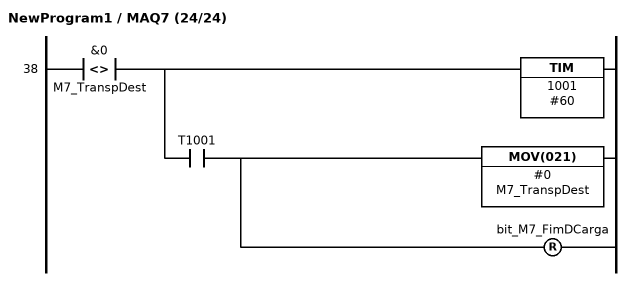
; [picture p24: NewProgram1 / MAQ7, rungs 38-38]
; rung 38
LD<>(305) &0 M7_TranspDest
TIM 1001 #60
AND T1001
MOV(021) #0 M7_TranspDest
RSET bit_M7_FimDCarga

### Section MAQ8

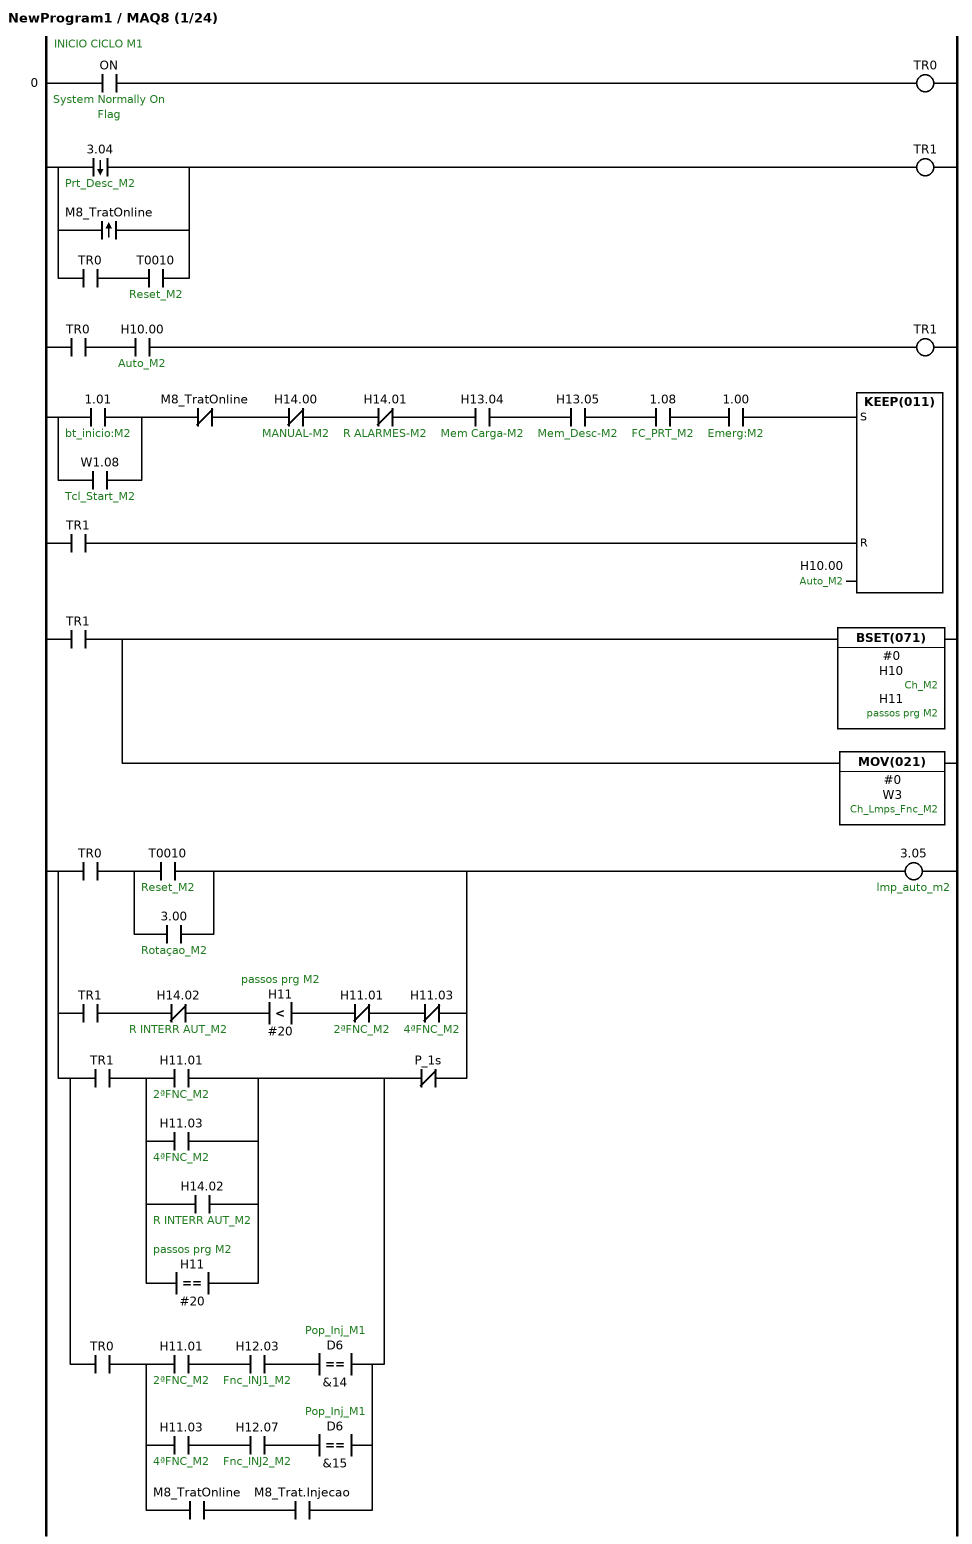
; rung 0: INICIO CICLO M1
LD 1.01  ; bt_inicio:M2
OR W1.08  ; Tcl_Start_M2
ANDNOT M8_TratOnline
ANDNOT H14.00  ; MANUAL-M2
ANDNOT H14.01  ; R ALARMES-M2
AND H13.04  ; Mem Carga-M2
AND H13.05  ; Mem_Desc-M2
AND 1.08  ; FC_PRT_M2
AND 1.00  ; Emerg:M2
%LD 3.04  ; Prt_Desc_M2
@OR M8_TratOnline
LD ON  ; System Normally On Flag
OUT TR0
AND T0010  ; Reset_M2
ORLD
OUT TR1
KEEP(011) H10.00  ; Auto_M2
LD TR1
BSET(071) #0 H10 H11  ; Ch_M2, passos prg M2
MOV(021) #0 W3  ; Ch_Lmps_Fnc_M2
LD TR0
LD T0010  ; Reset_M2
OR 3.00  ; Rotaçao_M2
ANDLD
LD TR0
AND H10.00  ; Auto_M2
OUT TR1
ANDNOT H14.02  ; R INTERR AUT_M2
AND<(310) H11 #20  ; passos prg M2
ANDNOT H11.01  ; 2ªFNC_M2
ANDNOT H11.03  ; 4ªFNC_M2
ORLD
LD TR1
LD H11.01  ; 2ªFNC_M2
OR H11.03  ; 4ªFNC_M2
OR H14.02  ; R INTERR AUT_M2
OR=(300) H11 #20  ; passos prg M2
ANDLD
LD TR0
LD H11.01  ; 2ªFNC_M2
AND H12.03  ; Fnc_INJ1_M2
AND=(300) D6 &14  ; Pop_Inj_M1
LD H11.03  ; 4ªFNC_M2
AND H12.07  ; Fnc_INJ2_M2
AND=(300) D6 &15  ; Pop_Inj_M1
ORLD
LD M8_TratOnline
AND M8_Trat.Injecao
ORLD
ANDLD
ORLD
ANDNOT P_1s
ORLD
OUT 3.05  ; lmp_auto_m2

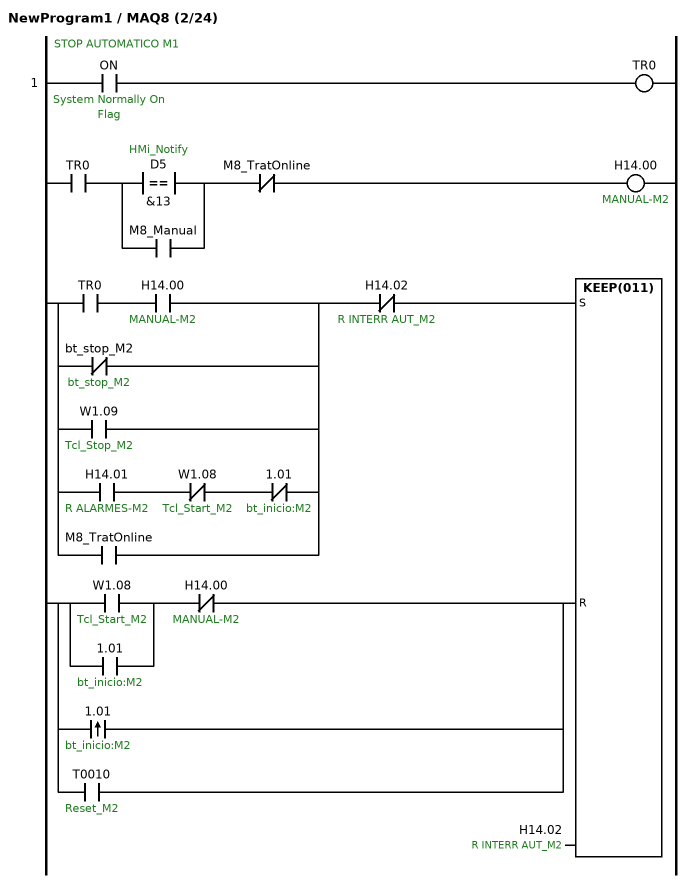
; rung 1: STOP AUTOMATICO M1
LD ON  ; System Normally On Flag
OUT TR0
LD=L(301) D5 &13  ; HMi_Notify
OR M8_Manual
ANDLD
ANDNOT M8_TratOnline
OUT H14.00  ; MANUAL-M2
LD TR0
AND H14.00  ; MANUAL-M2
LDNOT bt_stop_M2  ; bt_stop_M2
OR W1.09  ; Tcl_Stop_M2
LD H14.01  ; R ALARMES-M2
ANDNOT W1.08  ; Tcl_Start_M2
ANDNOT 1.01  ; bt_inicio:M2
ORLD
OR M8_TratOnline
ORLD
ANDNOT H14.02  ; R INTERR AUT_M2
LD W1.08  ; Tcl_Start_M2
OR 1.01  ; bt_inicio:M2
ANDNOT H14.00  ; MANUAL-M2
@OR 1.01  ; bt_inicio:M2
OR T0010  ; Reset_M2
KEEP(011) H14.02  ; R INTERR AUT_M2

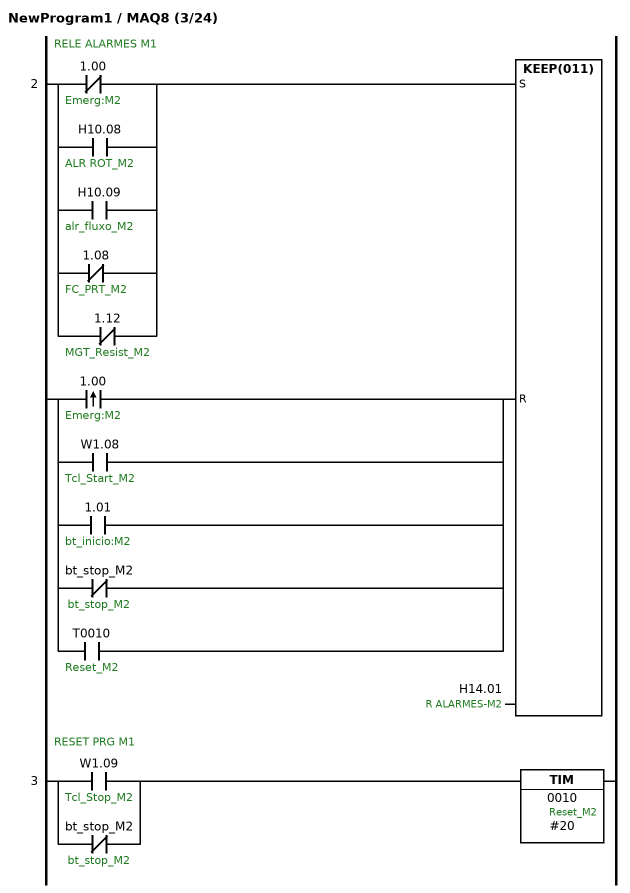
; rung 2: RELE ALARMES M1
LDNOT 1.00  ; Emerg:M2
OR H10.08  ; ALR ROT_M2
OR H10.09  ; alr_fluxo_M2
ORNOT 1.08  ; FC_PRT_M2
ORNOT 1.12  ; MGT_Resist_M2
@LD 1.00  ; Emerg:M2
OR W1.08  ; Tcl_Start_M2
OR 1.01  ; bt_inicio:M2
ORNOT bt_stop_M2  ; bt_stop_M2
OR T0010  ; Reset_M2
KEEP(011) H14.01  ; R ALARMES-M2
; rung 3: RESET PRG M1
LD W1.09  ; Tcl_Stop_M2
ORNOT bt_stop_M2  ; bt_stop_M2
TIM 0010 #20  ; Reset_M2

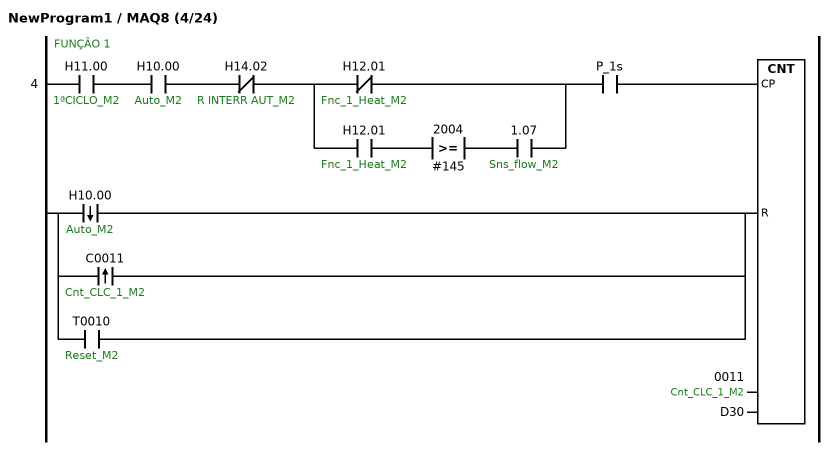
; rung 4: FUNÇÂO 1
LD H11.00  ; 1ªCICLO_M2
AND H10.00  ; Auto_M2
ANDNOT H14.02  ; R INTERR AUT_M2
LDNOT H12.01  ; Fnc_1_Heat_M2
LD H12.01  ; Fnc_1_Heat_M2
AND>=(325) 2004 #145
AND 1.07  ; Sns_flow_M2
ORLD
ANDLD
AND P_1s
%LD H10.00  ; Auto_M2
@OR C0011  ; Cnt_CLC_1_M2
OR T0010  ; Reset_M2
CNT 0011 D30  ; Cnt_CLC_1_M2

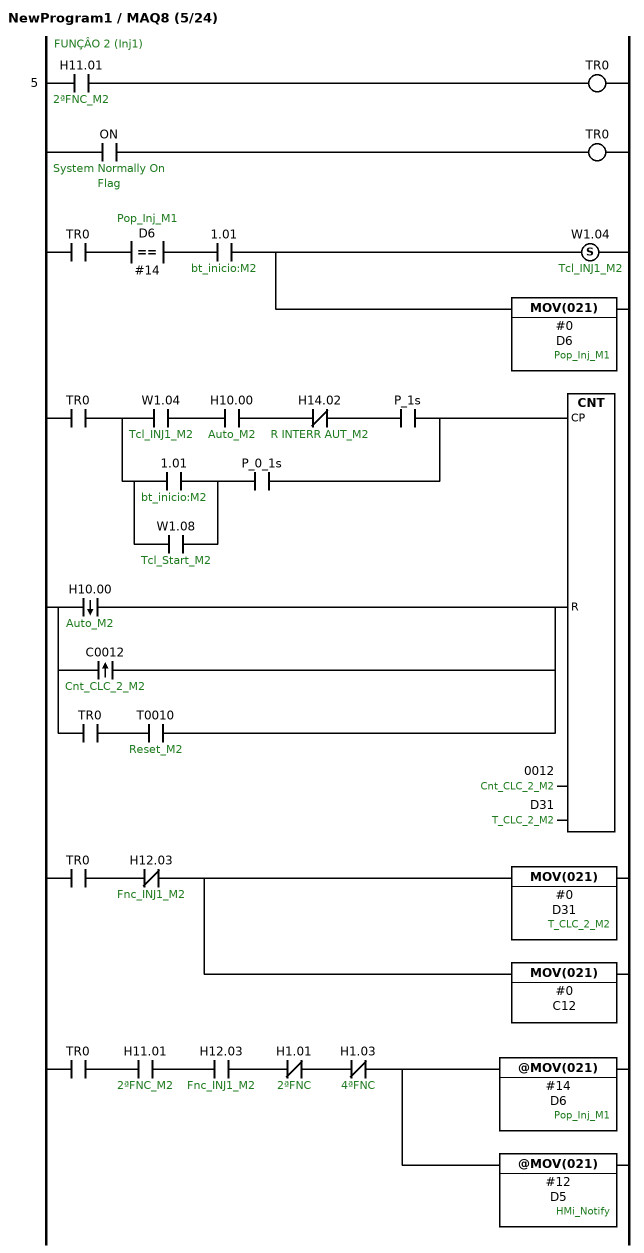
; rung 5: FUNÇÂO 2 (Inj1)
LD H11.01  ; 2ªFNC_M2
OUT TR0
AND=(300) D6 #14  ; Pop_Inj_M1
AND 1.01  ; bt_inicio:M2
SET W1.04  ; Tcl_INJ1_M2
MOV(021) #0 D6  ; Pop_Inj_M1
LD TR0
LD W1.04  ; Tcl_INJ1_M2
AND H10.00  ; Auto_M2
ANDNOT H14.02  ; R INTERR AUT_M2
AND P_1s
LD 1.01  ; bt_inicio:M2
OR W1.08  ; Tcl_Start_M2
AND P_0_1s
ORLD
ANDLD
%LD H10.00  ; Auto_M2
@OR C0012  ; Cnt_CLC_2_M2
LD ON  ; System Normally On Flag
OUT TR0
AND T0010  ; Reset_M2
ORLD
CNT 0012 D31  ; T_CLC_2_M2, Cnt_CLC_2_M2
LD TR0
ANDNOT H12.03  ; Fnc_INJ1_M2
MOV(021) #0 D31  ; T_CLC_2_M2
MOV(021) #0 C12
LD TR0
AND H11.01  ; 2ªFNC_M2
AND H12.03  ; Fnc_INJ1_M2
ANDNOT H1.01  ; 2ªFNC
ANDNOT H1.03  ; 4ªFNC
@MOV(021) #14 D6  ; Pop_Inj_M1
@MOV(021) #12 D5  ; HMi_Notify

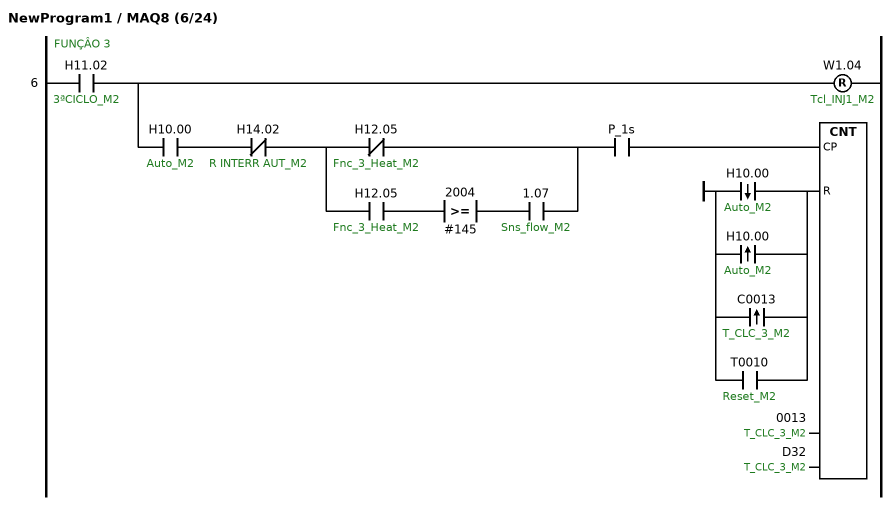
; rung 6: FUNÇÂO 3
LD H11.02  ; 3ªCICLO_M2
RSET W1.04  ; Tcl_INJ1_M2
AND H10.00  ; Auto_M2
ANDNOT H14.02  ; R INTERR AUT_M2
LDNOT H12.05  ; Fnc_3_Heat_M2
LD H12.05  ; Fnc_3_Heat_M2
AND>=(325) 2004 #145
AND 1.07  ; Sns_flow_M2
ORLD
ANDLD
AND P_1s
%LD H10.00  ; Auto_M2
@OR H10.00  ; Auto_M2
@OR C0013  ; T_CLC_3_M2
OR T0010  ; Reset_M2
CNT 0013 D32  ; T_CLC_3_M2

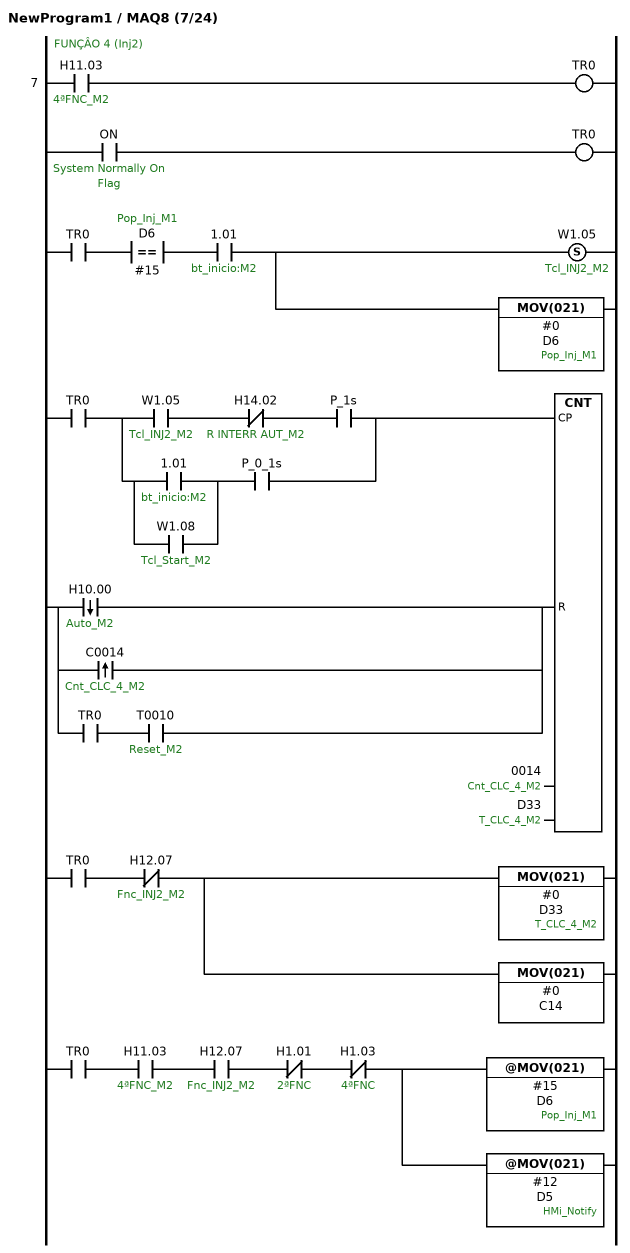
; rung 7: FUNÇÂO 4 (Inj2)
LD H11.03  ; 4ªFNC_M2
OUT TR0
AND=(300) D6 #15  ; Pop_Inj_M1
AND 1.01  ; bt_inicio:M2
SET W1.05  ; Tcl_INJ2_M2
MOV(021) #0 D6  ; Pop_Inj_M1
LD TR0
LD W1.05  ; Tcl_INJ2_M2
ANDNOT H14.02  ; R INTERR AUT_M2
AND P_1s
LD 1.01  ; bt_inicio:M2
OR W1.08  ; Tcl_Start_M2
AND P_0_1s
ORLD
ANDLD
%LD H10.00  ; Auto_M2
@OR C0014  ; Cnt_CLC_4_M2
LD ON  ; System Normally On Flag
OUT TR0
AND T0010  ; Reset_M2
ORLD
CNT 0014 D33  ; T_CLC_4_M2, Cnt_CLC_4_M2
LD TR0
ANDNOT H12.07  ; Fnc_INJ2_M2
MOV(021) #0 D33  ; T_CLC_4_M2
MOV(021) #0 C14
LD TR0
AND H11.03  ; 4ªFNC_M2
AND H12.07  ; Fnc_INJ2_M2
ANDNOT H1.01  ; 2ªFNC
ANDNOT H1.03  ; 4ªFNC
@MOV(021) #15 D6  ; Pop_Inj_M1
@MOV(021) #12 D5  ; HMi_Notify

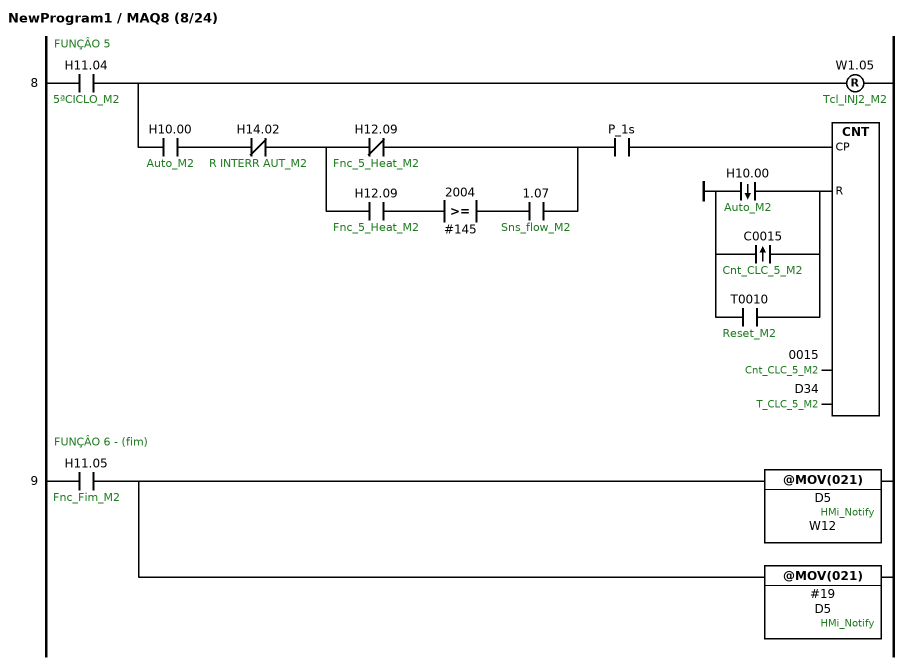
; rung 8: FUNÇÂO 5
LD H11.04  ; 5ªCICLO_M2
RSET W1.05  ; Tcl_INJ2_M2
AND H10.00  ; Auto_M2
ANDNOT H14.02  ; R INTERR AUT_M2
LDNOT H12.09  ; Fnc_5_Heat_M2
LD H12.09  ; Fnc_5_Heat_M2
AND>=(325) 2004 #145
AND 1.07  ; Sns_flow_M2
ORLD
ANDLD
AND P_1s
%LD H10.00  ; Auto_M2
@OR C0015  ; Cnt_CLC_5_M2
OR T0010  ; Reset_M2
CNT 0015 D34  ; T_CLC_5_M2, Cnt_CLC_5_M2
; rung 9: FUNÇÂO 6 - (fim)
LD H11.05  ; Fnc_Fim_M2
@MOV(021) D5 W12  ; HMi_Notify
@MOV(021) #19 D5  ; HMi_Notify

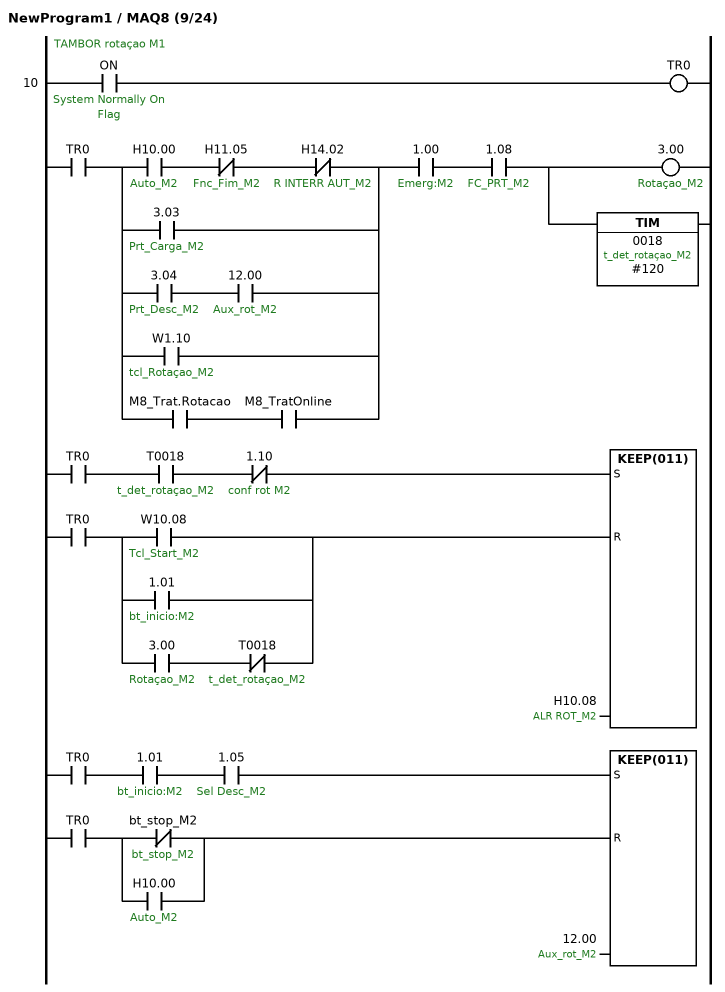
; rung 10: TAMBOR rotaçao M1
LD ON  ; System Normally On Flag
OUT TR0
LD H10.00  ; Auto_M2
ANDNOT H11.05  ; Fnc_Fim_M2
ANDNOT H14.02  ; R INTERR AUT_M2
OR 3.03  ; Prt_Carga_M2
LD 3.04  ; Prt_Desc_M2
AND 12.00  ; Aux_rot_M2
ORLD
OR W1.10  ; tcl_Rotaçao_M2
LD M8_Trat.Rotacao
AND M8_TratOnline
ORLD
ANDLD
AND 1.00  ; Emerg:M2
AND 1.08  ; FC_PRT_M2
OUT 3.00  ; Rotaçao_M2
TIM 0018 #120  ; t_det_rotaçao_M2
LD TR0
AND T0018  ; t_det_rotaçao_M2
ANDNOT 1.10  ; conf rot M2
LD TR0
LD W10.08  ; Tcl_Start_M2
OR 1.01  ; bt_inicio:M2
LD 3.00  ; Rotaçao_M2
ANDNOT T0018  ; t_det_rotaçao_M2
ORLD
ANDLD
KEEP(011) H10.08  ; ALR ROT_M2
LD TR0
AND 1.01  ; bt_inicio:M2
AND 1.05  ; Sel Desc_M2
LD TR0
LDNOT bt_stop_M2  ; bt_stop_M2
OR H10.00  ; Auto_M2
ANDLD
KEEP(011) 12.00  ; Aux_rot_M2

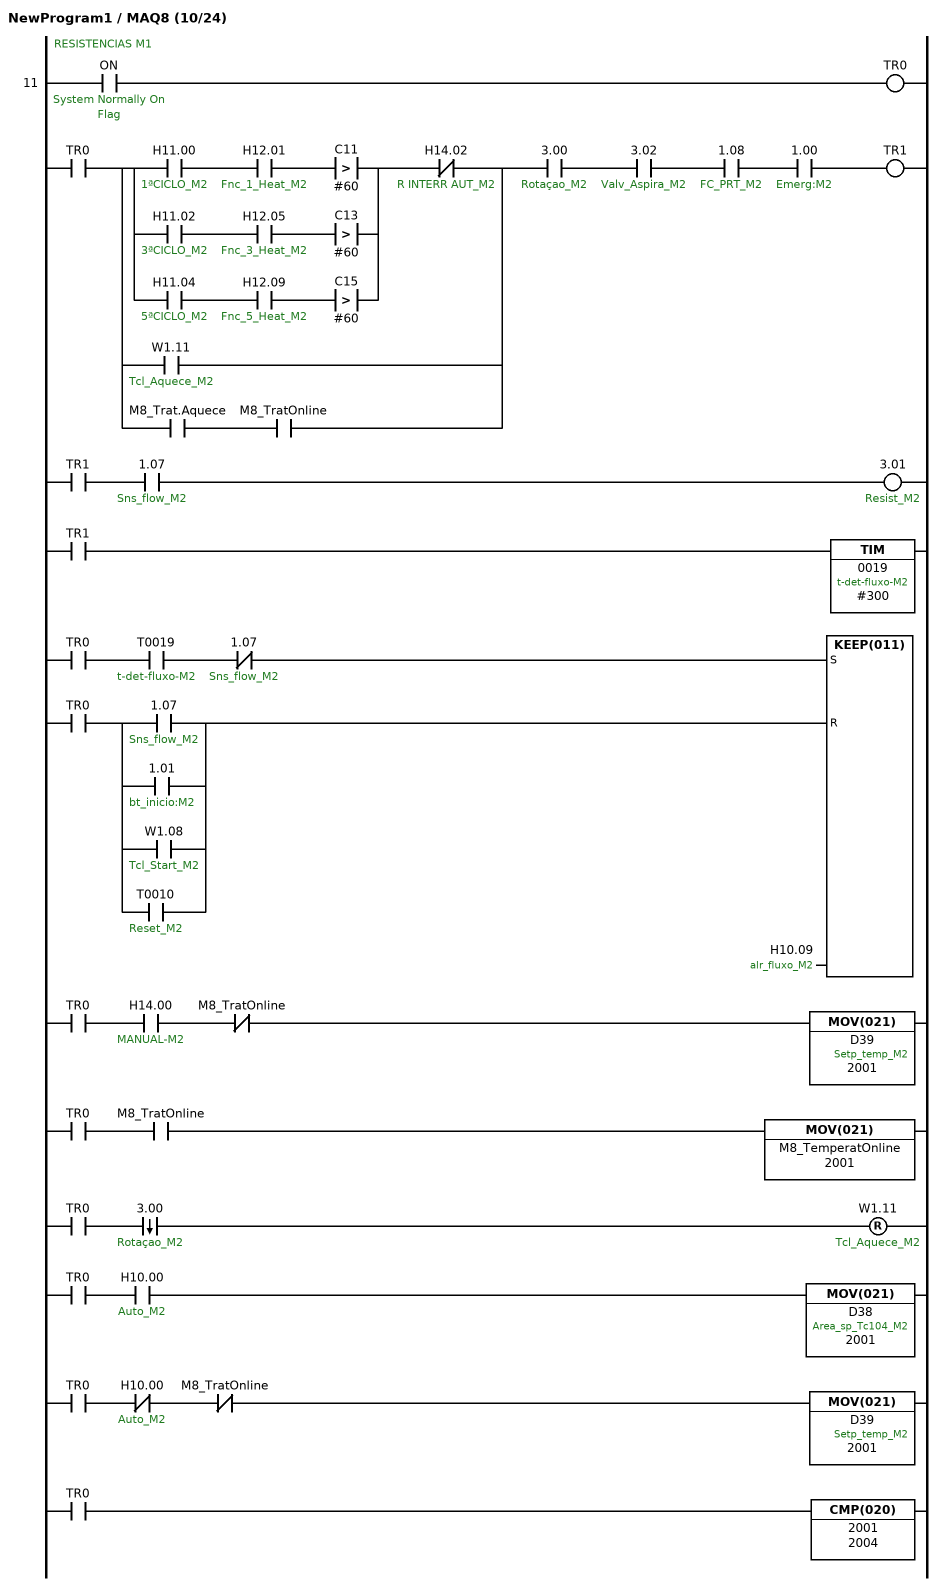
; rung 11: RESISTENCIAS M1
LD ON  ; System Normally On Flag
OUT TR0
LD H11.00  ; 1ªCICLO_M2
AND H12.01  ; Fnc_1_Heat_M2
AND>(320) C11 #60
LD H11.02  ; 3ªCICLO_M2
AND H12.05  ; Fnc_3_Heat_M2
AND>(320) C13 #60
ORLD
LD H11.04  ; 5ªCICLO_M2
AND H12.09  ; Fnc_5_Heat_M2
AND>(320) C15 #60
ORLD
ANDNOT H14.02  ; R INTERR AUT_M2
OR W1.11  ; Tcl_Aquece_M2
LD M8_Trat.Aquece
AND M8_TratOnline
ORLD
ANDLD
AND 3.00  ; Rotaçao_M2
AND 3.02  ; Valv_Aspira_M2
AND 1.08  ; FC_PRT_M2
AND 1.00  ; Emerg:M2
OUT TR1
AND 1.07  ; Sns_flow_M2
OUT 3.01  ; Resist_M2
LD TR1
TIM 0019 #300  ; t-det-fluxo-M2
LD TR0
AND T0019  ; t-det-fluxo-M2
ANDNOT 1.07  ; Sns_flow_M2
LD TR0
LD 1.07  ; Sns_flow_M2
OR 1.01  ; bt_inicio:M2
OR W1.08  ; Tcl_Start_M2
OR T0010  ; Reset_M2
ANDLD
KEEP(011) H10.09  ; alr_fluxo_M2
LD TR0
AND H14.00  ; MANUAL-M2
ANDNOT M8_TratOnline
MOV(021) D39 2001  ; Setp_temp_M2
LD TR0
AND M8_TratOnline
MOV(021) M8_TemperatOnline 2001
LD TR0
%AND 3.00  ; Rotaçao_M2
RSET W1.11  ; Tcl_Aquece_M2
LD TR0
AND H10.00  ; Auto_M2
MOV(021) D38 2001  ; Area_sp_Tc104_M2
LD TR0
ANDNOT H10.00  ; Auto_M2
ANDNOT M8_TratOnline
MOV(021) D39 2001  ; Setp_temp_M2
LD TR0
CMP(020) 2001 2004

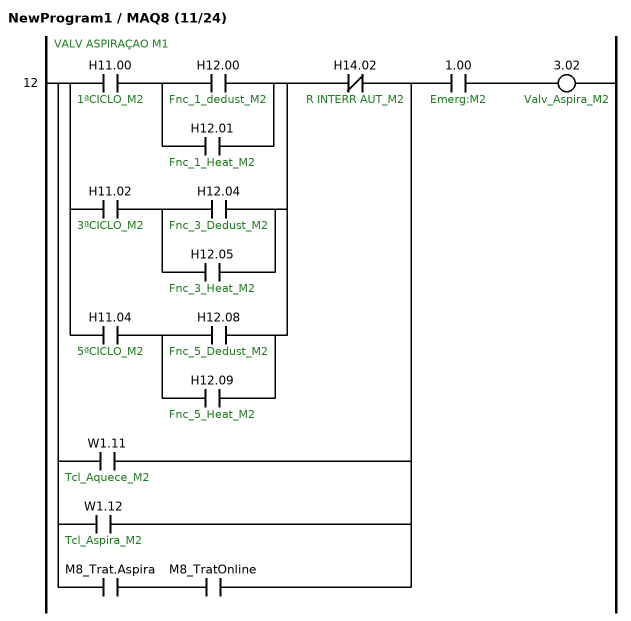
; rung 12: VALV ASPIRAÇAO M1
LD H11.00  ; 1ªCICLO_M2
LD H12.00  ; Fnc_1_dedust_M2
OR H12.01  ; Fnc_1_Heat_M2
ANDLD
LD H11.02  ; 3ªCICLO_M2
LD H12.04  ; Fnc_3_Dedust_M2
OR H12.05  ; Fnc_3_Heat_M2
ANDLD
ORLD
LD H11.04  ; 5ªCICLO_M2
LD H12.08  ; Fnc_5_Dedust_M2
OR H12.09  ; Fnc_5_Heat_M2
ANDLD
ORLD
ANDNOT H14.02  ; R INTERR AUT_M2
OR W1.11  ; Tcl_Aquece_M2
OR W1.12  ; Tcl_Aspira_M2
LD M8_Trat.Aspira
AND M8_TratOnline
ORLD
AND 1.00  ; Emerg:M2
OUT 3.02  ; Valv_Aspira_M2

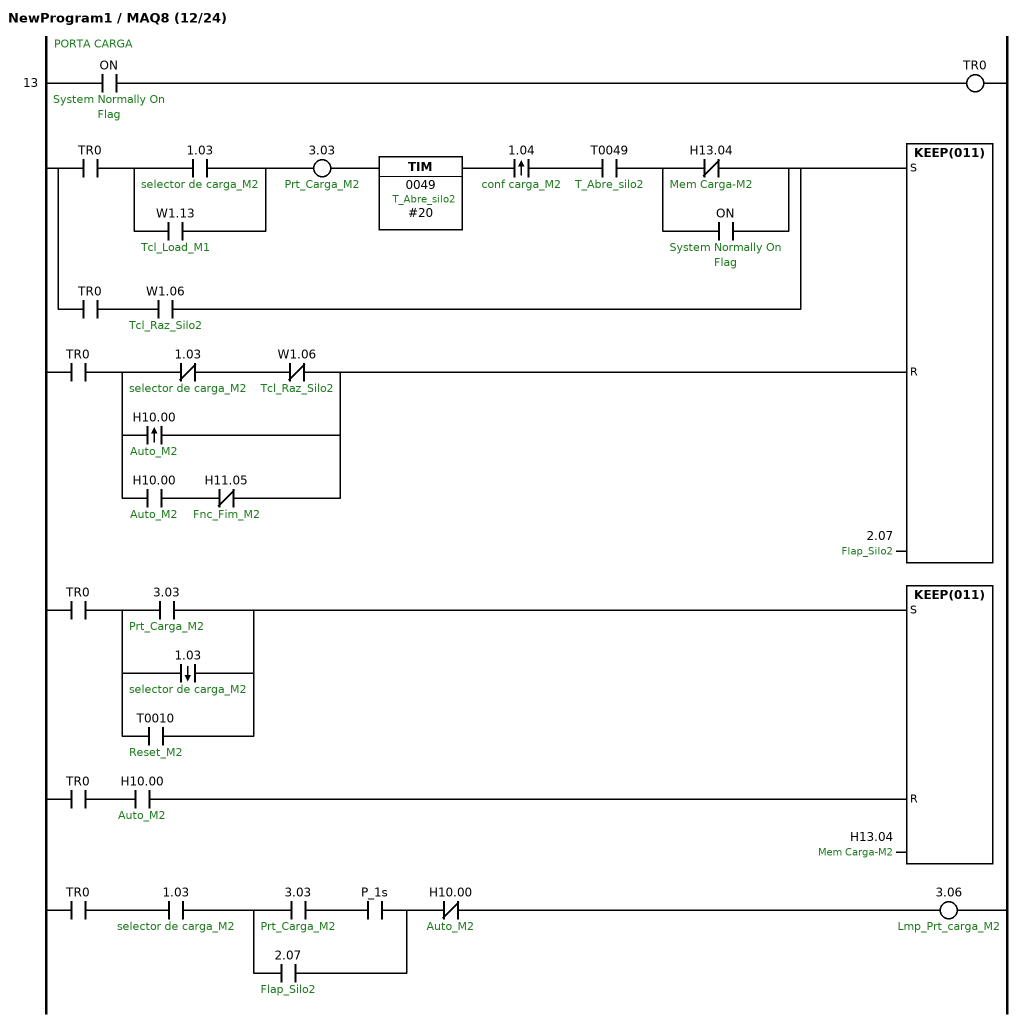
; rung 13: PORTA CARGA
LD ON  ; System Normally On Flag
OUT TR0
LD 1.03  ; selector de carga_M2
OR W1.13  ; Tcl_Load_M1
ANDLD
OUT 3.03  ; Prt_Carga_M2
TIM 0049 #20  ; T_Abre_silo2
@AND 1.04  ; conf carga_M2
AND T0049  ; T_Abre_silo2
LDNOT H13.04  ; Mem Carga-M2
OR ON  ; System Normally On Flag
ANDLD
LD TR0
AND W1.06  ; Tcl_Raz_Silo2
ORLD
LD TR0
LDNOT 1.03  ; selector de carga_M2
ANDNOT W1.06  ; Tcl_Raz_Silo2
@OR H10.00  ; Auto_M2
LD H10.00  ; Auto_M2
ANDNOT H11.05  ; Fnc_Fim_M2
ORLD
ANDLD
KEEP(011) 2.07  ; Flap_Silo2
LD TR0
LD 3.03  ; Prt_Carga_M2
%OR 1.03  ; selector de carga_M2
OR T0010  ; Reset_M2
ANDLD
LD TR0
AND H10.00  ; Auto_M2
KEEP(011) H13.04  ; Mem Carga-M2
LD TR0
AND 1.03  ; selector de carga_M2
LD 3.03  ; Prt_Carga_M2
AND P_1s
OR 2.07  ; Flap_Silo2
ANDLD
ANDNOT H10.00  ; Auto_M2
OUT 3.06  ; Lmp_Prt_carga_M2

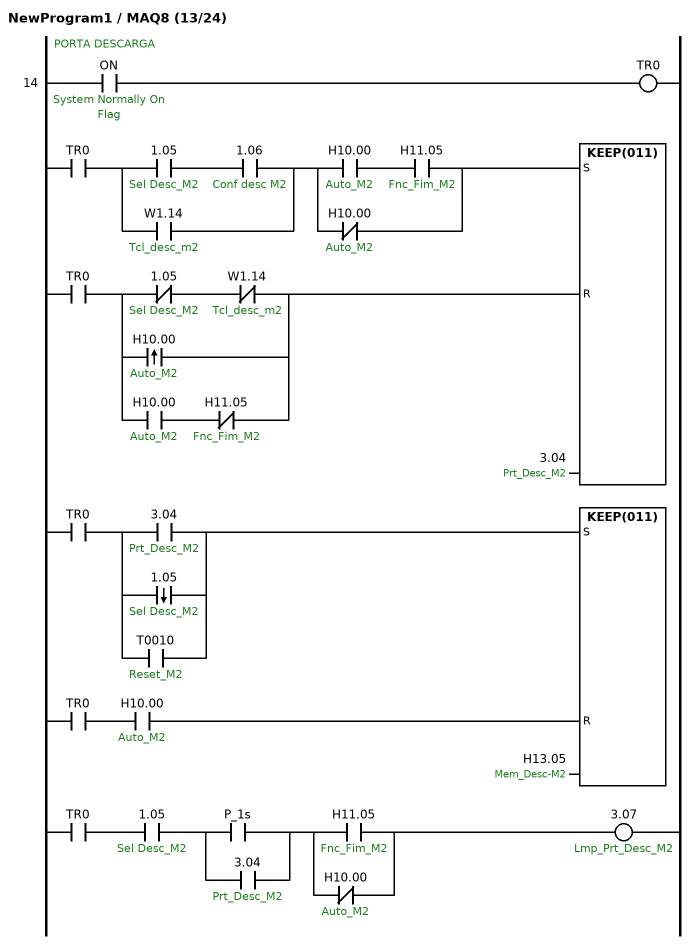
; rung 14: PORTA DESCARGA
LD ON  ; System Normally On Flag
OUT TR0
LD 1.05  ; Sel Desc_M2
AND 1.06  ; Conf desc M2
OR W1.14  ; Tcl_desc_m2
ANDLD
LD H10.00  ; Auto_M2
AND H11.05  ; Fnc_Fim_M2
ORNOT H10.00  ; Auto_M2
ANDLD
LD TR0
LDNOT 1.05  ; Sel Desc_M2
ANDNOT W1.14  ; Tcl_desc_m2
@OR H10.00  ; Auto_M2
LD H10.00  ; Auto_M2
ANDNOT H11.05  ; Fnc_Fim_M2
ORLD
ANDLD
KEEP(011) 3.04  ; Prt_Desc_M2
LD TR0
LD 3.04  ; Prt_Desc_M2
%OR 1.05  ; Sel Desc_M2
OR T0010  ; Reset_M2
ANDLD
LD TR0
AND H10.00  ; Auto_M2
KEEP(011) H13.05  ; Mem_Desc-M2
LD TR0
AND 1.05  ; Sel Desc_M2
LD P_1s
OR 3.04  ; Prt_Desc_M2
ANDLD
LD H11.05  ; Fnc_Fim_M2
ORNOT H10.00  ; Auto_M2
ANDLD
OUT 3.07  ; Lmp_Prt_Desc_M2

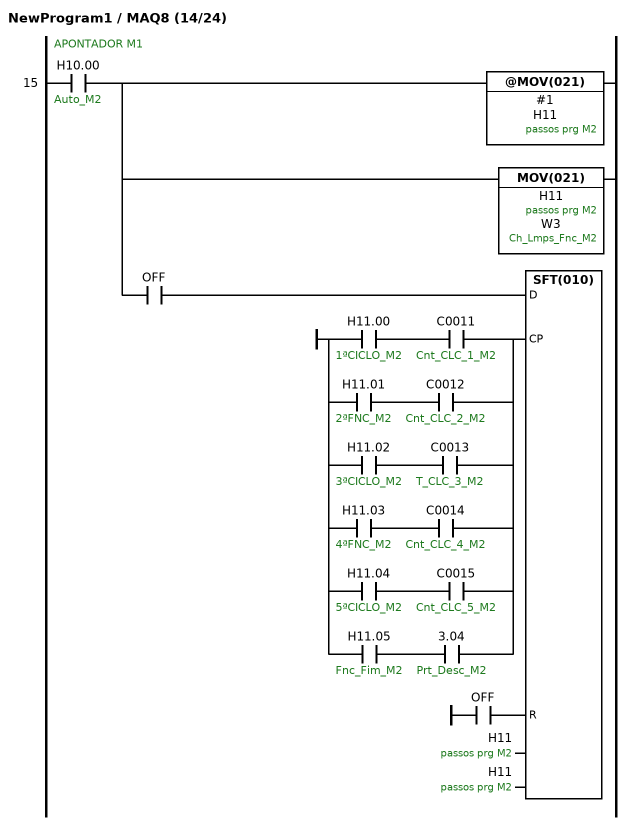
; rung 15: APONTADOR M1
LD H10.00  ; Auto_M2
@MOV(021) #1 H11  ; passos prg M2
MOV(021) H11 W3  ; passos prg M2, Ch_Lmps_Fnc_M2
AND OFF
LD H11.00  ; 1ªCICLO_M2
AND C0011  ; Cnt_CLC_1_M2
LD H11.01  ; 2ªFNC_M2
AND C0012  ; Cnt_CLC_2_M2
ORLD
LD H11.02  ; 3ªCICLO_M2
AND C0013  ; T_CLC_3_M2
ORLD
LD H11.03  ; 4ªFNC_M2
AND C0014  ; Cnt_CLC_4_M2
ORLD
LD H11.04  ; 5ªCICLO_M2
AND C0015  ; Cnt_CLC_5_M2
ORLD
LD H11.05  ; Fnc_Fim_M2
AND 3.04  ; Prt_Desc_M2
ORLD
LD OFF
SFT(010) H11 H11  ; passos prg M2

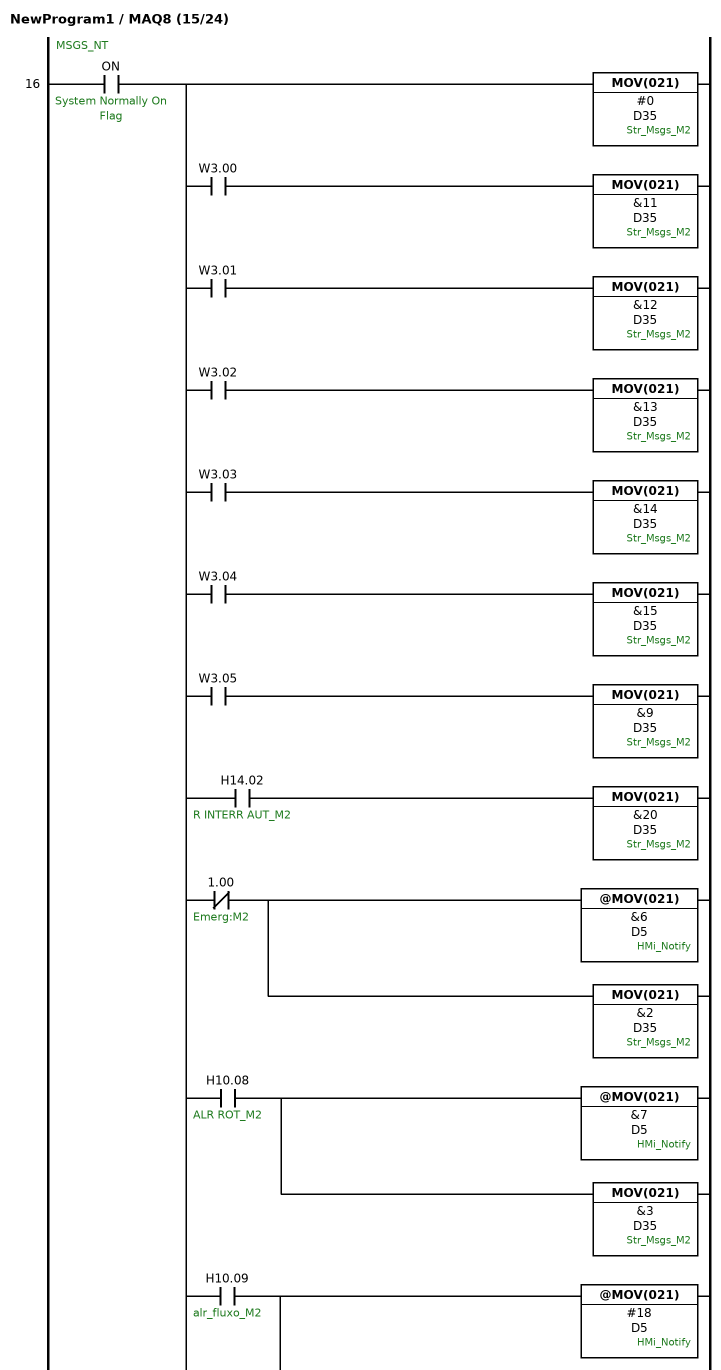

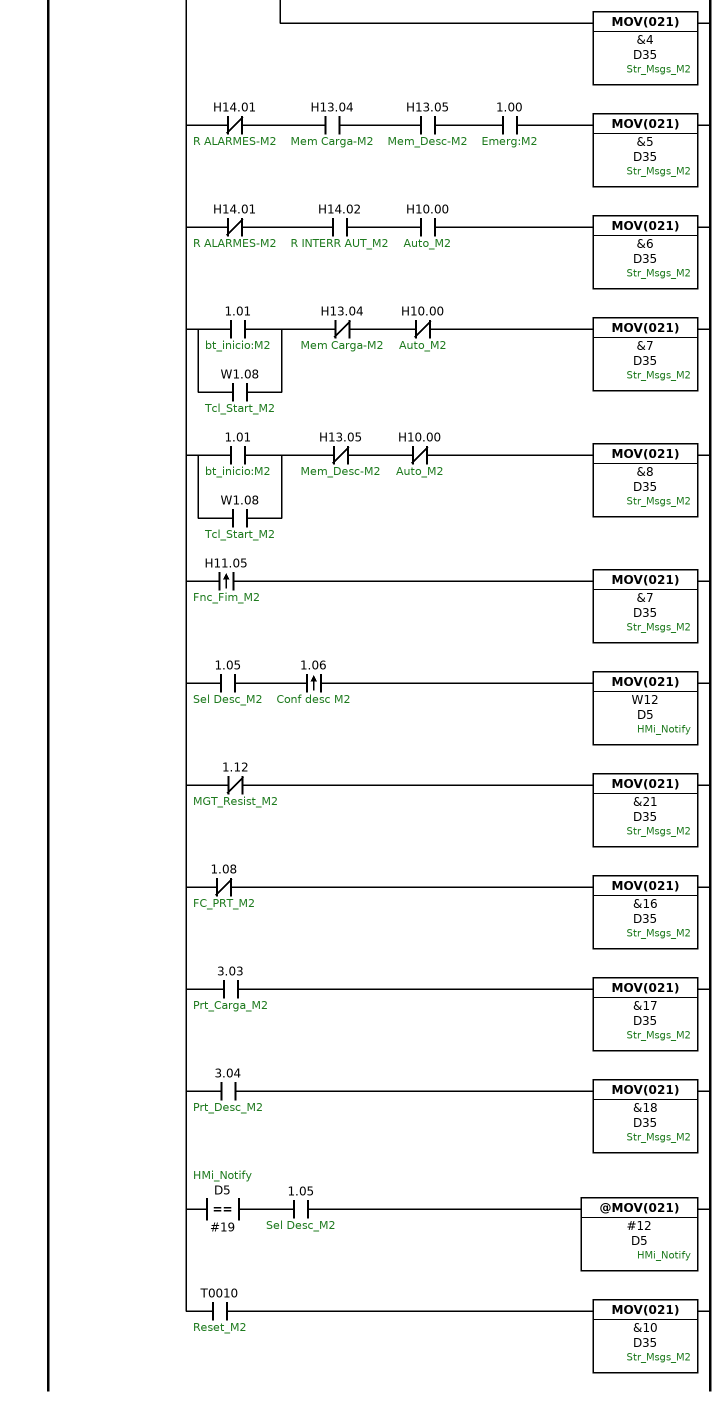
; rung 16: MSGS_NT
LD ON  ; System Normally On Flag
OUT TR0
MOV(021) #0 D35  ; Str_Msgs_M2
AND W3.00
MOV(021) &11 D35  ; Str_Msgs_M2
LD TR0
AND W3.01
MOV(021) &12 D35  ; Str_Msgs_M2
LD TR0
AND W3.02
MOV(021) &13 D35  ; Str_Msgs_M2
LD TR0
AND W3.03
MOV(021) &14 D35  ; Str_Msgs_M2
LD TR0
AND W3.04
MOV(021) &15 D35  ; Str_Msgs_M2
LD TR0
AND W3.05
MOV(021) &9 D35  ; Str_Msgs_M2
LD TR0
AND H14.02  ; R INTERR AUT_M2
MOV(021) &20 D35  ; Str_Msgs_M2
LD TR0
ANDNOT 1.00  ; Emerg:M2
@MOV(021) &6 D5  ; HMi_Notify
MOV(021) &2 D35  ; Str_Msgs_M2
LD TR0
AND H10.08  ; ALR ROT_M2
@MOV(021) &7 D5  ; HMi_Notify
MOV(021) &3 D35  ; Str_Msgs_M2
LD TR0
AND H10.09  ; alr_fluxo_M2
@MOV(021) #18 D5  ; HMi_Notify
MOV(021) &4 D35  ; Str_Msgs_M2
LD TR0
ANDNOT H14.01  ; R ALARMES-M2
AND H13.04  ; Mem Carga-M2
AND H13.05  ; Mem_Desc-M2
AND 1.00  ; Emerg:M2
MOV(021) &5 D35  ; Str_Msgs_M2
LD TR0
ANDNOT H14.01  ; R ALARMES-M2
AND H14.02  ; R INTERR AUT_M2
AND H10.00  ; Auto_M2
MOV(021) &6 D35  ; Str_Msgs_M2
LD TR0
LD 1.01  ; bt_inicio:M2
OR W1.08  ; Tcl_Start_M2
ANDLD
ANDNOT H13.04  ; Mem Carga-M2
ANDNOT H10.00  ; Auto_M2
MOV(021) &7 D35  ; Str_Msgs_M2
LD TR0
LD 1.01  ; bt_inicio:M2
OR W1.08  ; Tcl_Start_M2
ANDLD
ANDNOT H13.05  ; Mem_Desc-M2
ANDNOT H10.00  ; Auto_M2
MOV(021) &8 D35  ; Str_Msgs_M2
LD TR0
@AND H11.05  ; Fnc_Fim_M2
MOV(021) &7 D35  ; Str_Msgs_M2
LD TR0
AND 1.05  ; Sel Desc_M2
@AND 1.06  ; Conf desc M2
MOV(021) W12 D5  ; HMi_Notify
LD TR0
ANDNOT 1.12  ; MGT_Resist_M2
MOV(021) &21 D35  ; Str_Msgs_M2
LD TR0
ANDNOT 1.08  ; FC_PRT_M2
MOV(021) &16 D35  ; Str_Msgs_M2
LD TR0
AND 3.03  ; Prt_Carga_M2
MOV(021) &17 D35  ; Str_Msgs_M2
LD TR0
AND 3.04  ; Prt_Desc_M2
MOV(021) &18 D35  ; Str_Msgs_M2
LD TR0
AND=(300) D5 #19  ; HMi_Notify
AND 1.05  ; Sel Desc_M2
@MOV(021) #12 D5  ; HMi_Notify
LD TR0
AND T0010  ; Reset_M2
MOV(021) &10 D35  ; Str_Msgs_M2

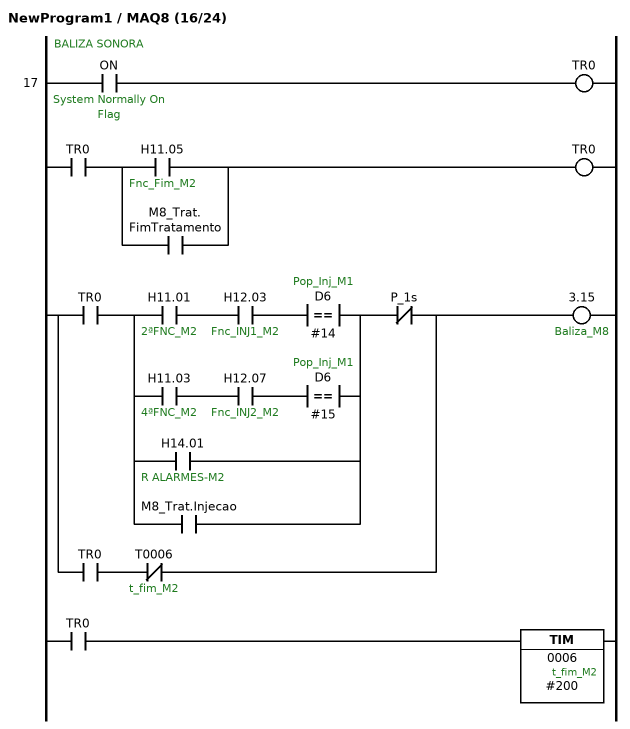
; rung 17: BALIZA SONORA
LD ON  ; System Normally On Flag
OUT TR0
LD H11.01  ; 2ªFNC_M2
AND H12.03  ; Fnc_INJ1_M2
AND=(300) D6 #14  ; Pop_Inj_M1
LD H11.03  ; 4ªFNC_M2
AND H12.07  ; Fnc_INJ2_M2
AND=(300) D6 #15  ; Pop_Inj_M1
ORLD
OR H14.01  ; R ALARMES-M2
OR M8_Trat.Injecao
ANDLD
ANDNOT P_1s
LD TR0
LD H11.05  ; Fnc_Fim_M2
OR M8_Trat.FimTratamento
ANDLD
OUT TR0
ANDNOT T0006  ; t_fim_M2
ORLD
OUT 3.15  ; Baliza_M8
LD TR0
TIM 0006 #200  ; t_fim_M2

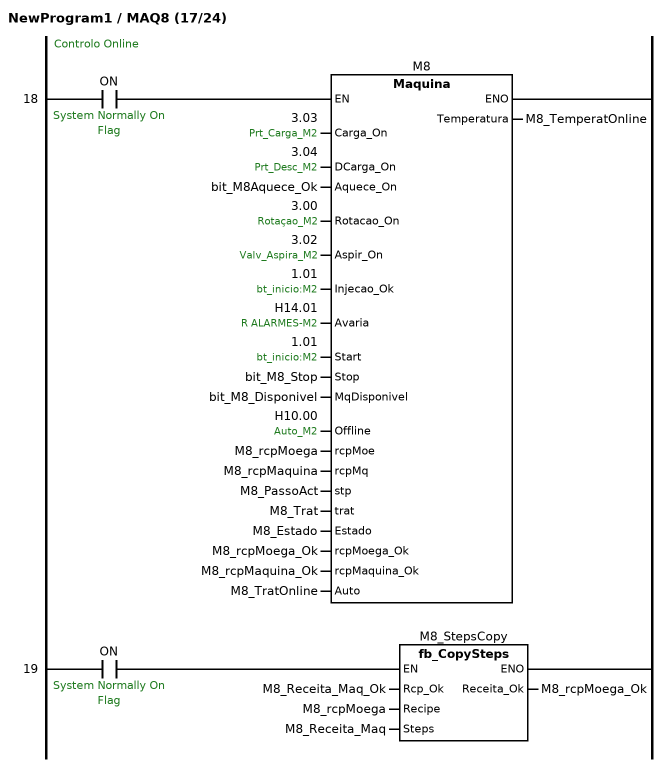
; rung 18: Controlo Online
LD ON  ; System Normally On Flag
CALL M8 : Maquina (Carga_On := 3.03, DCarga_On := 3.04, Aquece_On := bit_M8Aquece_Ok, Rotacao_On := 3.00, Aspir_On := 3.02, Injecao_Ok := 1.01, Avaria := H14.01, Start := 1.01, Stop := bit_M8_Stop, MqDisponivel := bit_M8_Disponivel, Offline := H10.00, rcpMoe := M8_rcpMoega, rcpMq := M8_rcpMaquina, stp := M8_PassoAct, trat := M8_Trat, Estado := M8_Estado, rcpMoega_Ok := M8_rcpMoega_Ok, rcpMaquina_Ok := M8_rcpMaquina_Ok, Auto := M8_TratOnline, Temperatura => M8_TemperatOnline)  ; Prt_Carga_M2, Prt_Desc_M2, Rotaçao_M2, Valv_Aspira_M2, bt_inicio:M2, R ALARMES-M2, Auto_M2
; rung 19
LD ON  ; System Normally On Flag
CALL M8_StepsCopy : fb_CopySteps (Rcp_Ok := M8_Receita_Maq_Ok, Recipe := M8_rcpMoega, Steps := M8_Receita_Maq, Receita_Ok => M8_rcpMoega_Ok)

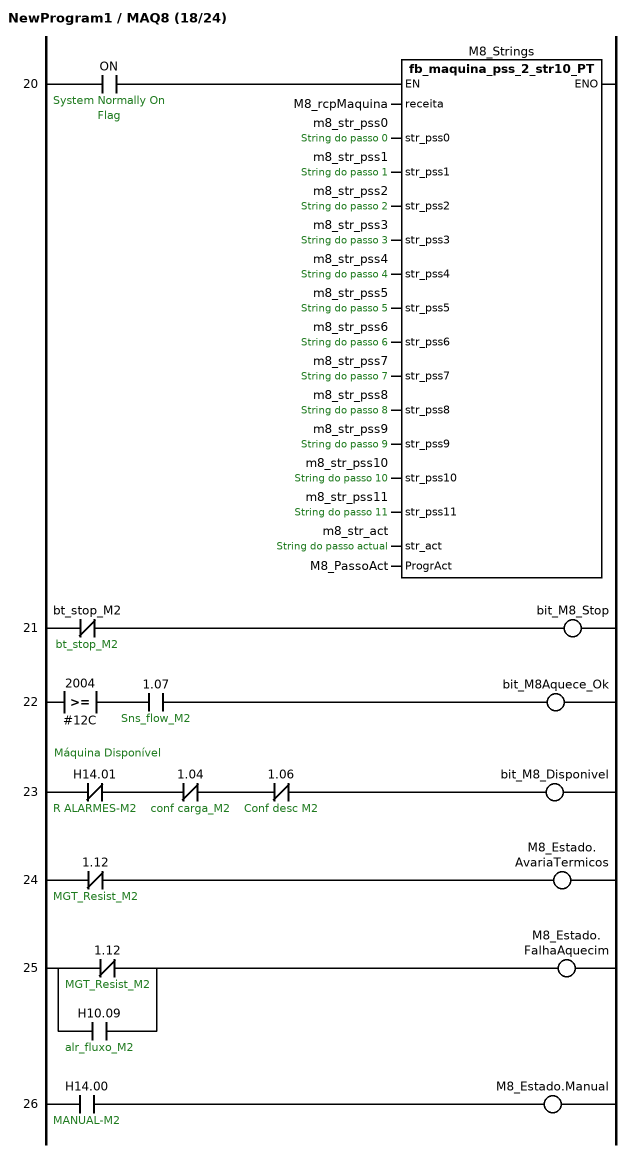
; rung 20
LD ON  ; System Normally On Flag
CALL M8_Strings : fb_maquina_pss_2_str10_PT (receita := M8_rcpMaquina, str_pss0 := m8_str_pss0, str_pss1 := m8_str_pss1, str_pss2 := m8_str_pss2, str_pss3 := m8_str_pss3, str_pss4 := m8_str_pss4, str_pss5 := m8_str_pss5, str_pss6 := m8_str_pss6, str_pss7 := m8_str_pss7, str_pss8 := m8_str_pss8, str_pss9 := m8_str_pss9, str_pss10 := m8_str_pss10, str_pss11 := m8_str_pss11, str_act := m8_str_act, ProgrAct := M8_PassoAct)  ; String do passo 0, String do passo 1, String do passo 2, String do passo 3, String do passo 4, String do passo 5, String do passo 6, String do passo 7, String do passo 8, String do passo 9, String do passo 10, String do passo 11, String do passo actual
; rung 21
LDNOT bt_stop_M2  ; bt_stop_M2
OUT bit_M8_Stop
; rung 22
LD>=(325) 2004 #12C
AND 1.07  ; Sns_flow_M2
OUT bit_M8Aquece_Ok
; rung 23: Máquina Disponível
LDNOT H14.01  ; R ALARMES-M2
ANDNOT 1.04  ; conf carga_M2
ANDNOT 1.06  ; Conf desc M2
OUT bit_M8_Disponivel
; rung 24
LDNOT 1.12  ; MGT_Resist_M2
OUT M8_Estado.AvariaTermicos
; rung 25
LDNOT 1.12  ; MGT_Resist_M2
OR H10.09  ; alr_fluxo_M2
OUT M8_Estado.FalhaAquecim
; rung 26
LD H14.00  ; MANUAL-M2
OUT M8_Estado.Manual

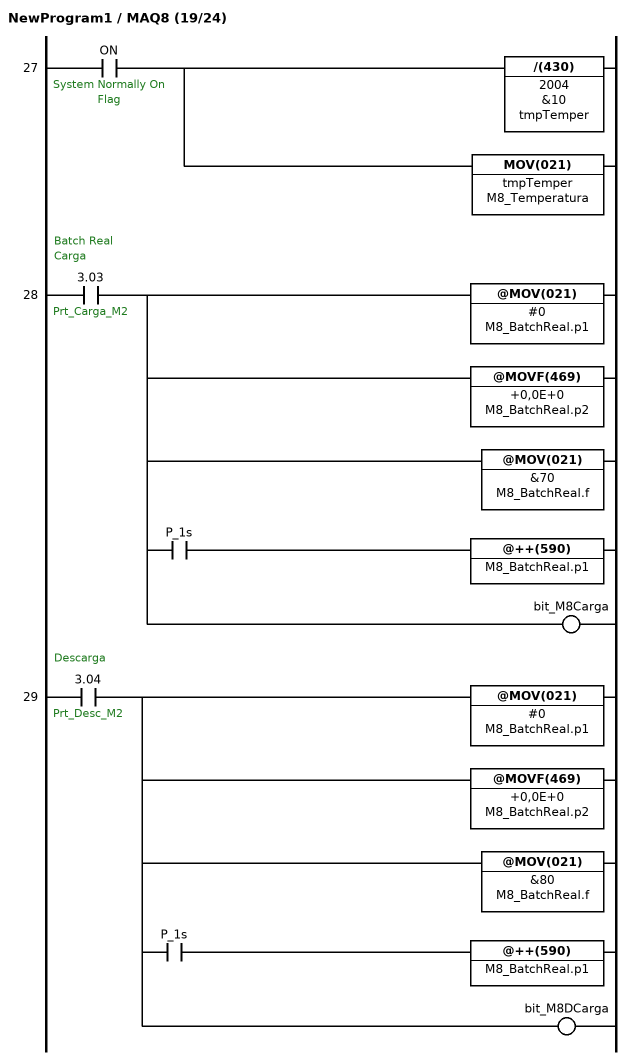
; rung 27
LD ON  ; System Normally On Flag
/(430) 2004 &10 tmpTemper
MOV(021) tmpTemper M8_Temperatura
; rung 28: Batch Real / Carga
LD 3.03  ; Prt_Carga_M2
OUT TR0
@MOV(021) #0 M8_BatchReal.p1
@MOVF(469) +0,0E+0 M8_BatchReal.p2
@MOV(021) &70 M8_BatchReal.f
AND P_1s
@++(590) M8_BatchReal.p1
LD TR0
OUT bit_M8Carga
; rung 29: Descarga
LD 3.04  ; Prt_Desc_M2
OUT TR0
@MOV(021) #0 M8_BatchReal.p1
@MOVF(469) +0,0E+0 M8_BatchReal.p2
@MOV(021) &80 M8_BatchReal.f
AND P_1s
@++(590) M8_BatchReal.p1
LD TR0
OUT bit_M8DCarga

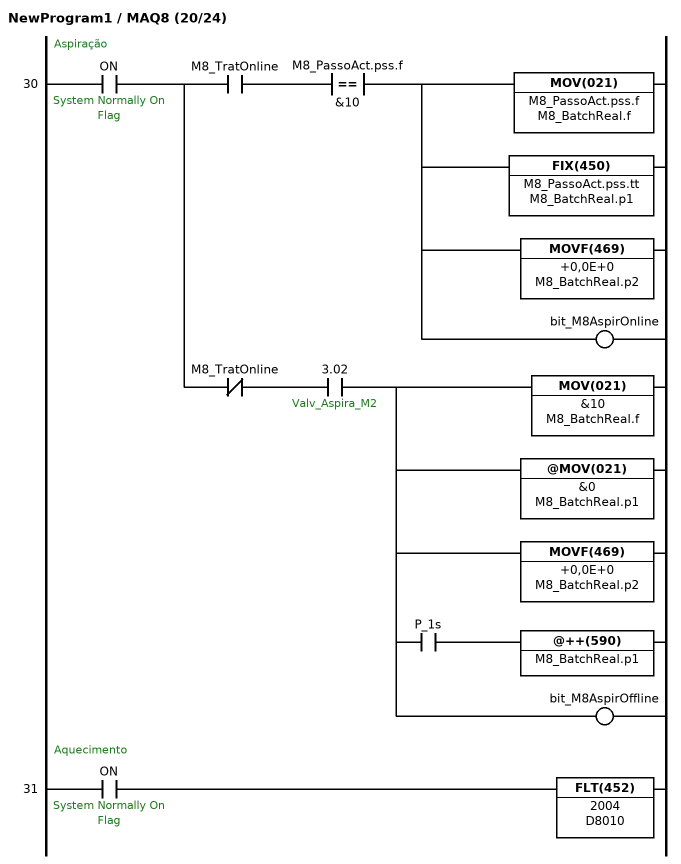
; rung 30: Aspiração
LD ON  ; System Normally On Flag
OUT TR0
AND M8_TratOnline
AND=(300) M8_PassoAct.pss.f &10
MOV(021) M8_PassoAct.pss.f M8_BatchReal.f
FIX(450) M8_PassoAct.pss.tt M8_BatchReal.p1
MOVF(469) +0,0E+0 M8_BatchReal.p2
OUT bit_M8AspirOnline
LD TR0
ANDNOT M8_TratOnline
AND 3.02  ; Valv_Aspira_M2
OUT TR0
MOV(021) &10 M8_BatchReal.f
@MOV(021) &0 M8_BatchReal.p1
MOVF(469) +0,0E+0 M8_BatchReal.p2
AND P_1s
@++(590) M8_BatchReal.p1
LD TR0
OUT bit_M8AspirOffline
; rung 31: Aquecimento
LD ON  ; System Normally On Flag
FLT(452) 2004 D8010

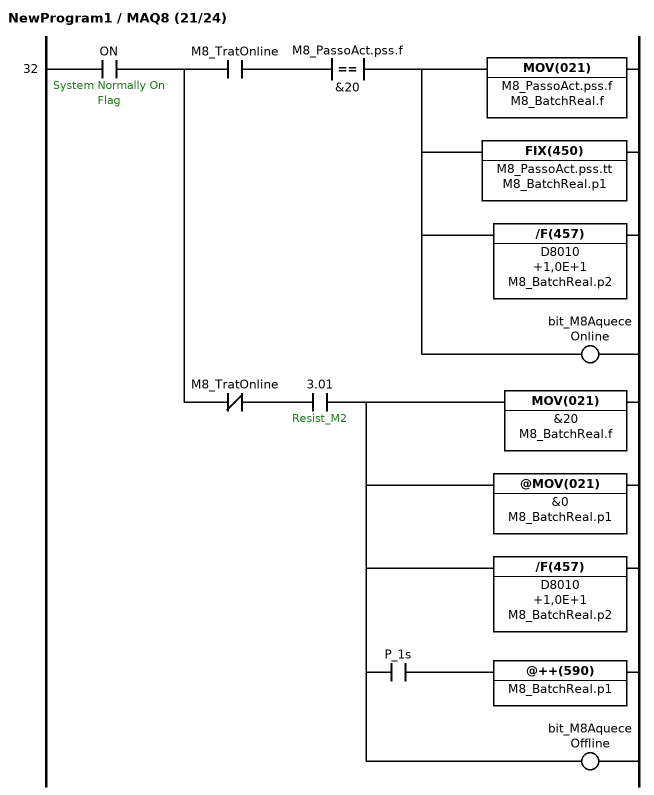
; rung 32
LD ON  ; System Normally On Flag
OUT TR0
AND M8_TratOnline
AND=(300) M8_PassoAct.pss.f &20
MOV(021) M8_PassoAct.pss.f M8_BatchReal.f
FIX(450) M8_PassoAct.pss.tt M8_BatchReal.p1
/F(457) D8010 +1,0E+1 M8_BatchReal.p2
OUT bit_M8AqueceOnline
LD TR0
ANDNOT M8_TratOnline
AND 3.01  ; Resist_M2
OUT TR0
MOV(021) &20 M8_BatchReal.f
@MOV(021) &0 M8_BatchReal.p1
/F(457) D8010 +1,0E+1 M8_BatchReal.p2
AND P_1s
@++(590) M8_BatchReal.p1
LD TR0
OUT bit_M8AqueceOffline

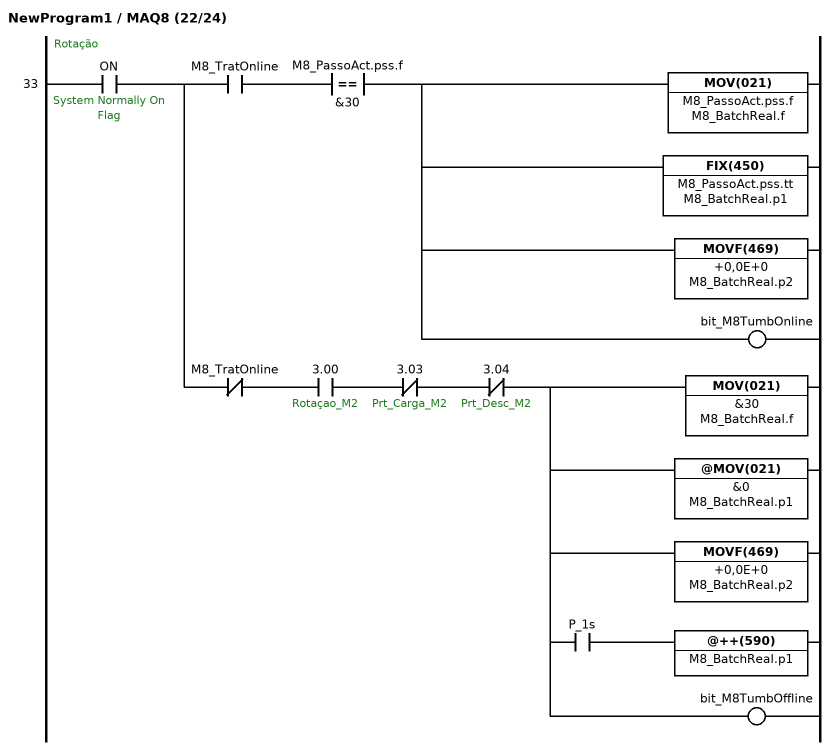
; rung 33: Rotação
LD ON  ; System Normally On Flag
OUT TR0
AND M8_TratOnline
AND=(300) M8_PassoAct.pss.f &30
MOV(021) M8_PassoAct.pss.f M8_BatchReal.f
FIX(450) M8_PassoAct.pss.tt M8_BatchReal.p1
MOVF(469) +0,0E+0 M8_BatchReal.p2
OUT bit_M8TumbOnline
LD TR0
ANDNOT M8_TratOnline
AND 3.00  ; Rotaçao_M2
ANDNOT 3.03  ; Prt_Carga_M2
ANDNOT 3.04  ; Prt_Desc_M2
OUT TR0
MOV(021) &30 M8_BatchReal.f
@MOV(021) &0 M8_BatchReal.p1
MOVF(469) +0,0E+0 M8_BatchReal.p2
AND P_1s
@++(590) M8_BatchReal.p1
LD TR0
OUT bit_M8TumbOffline

